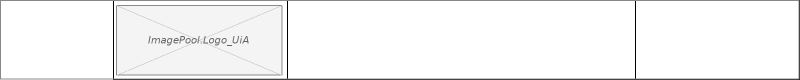
VISUALIZATION Header  // 800x80
    Rectangle (287,0 350x80), "MOTION LIMIT: OFF"
    Textfield (306,41 311x30), "TURN ON IN SETTINGS"
    Rectangle (113,0 175x80)
    Rectangle (287,0 350x80), invisible if: HMI.bBlink, input disabled if: HMI.bBlink
    Rectangle (635,0 165x80)
    Image (116,5 166x70), image: ImagePool.Logo_UiA
END_VISUALIZATION

(* stored: Version 1.1.0.1, ProductVersion 3.1.4024.12
   Visu Header: Id {86ca271f-4ae1-4eaa-9202-48f028a937e6} *)
